PROGRAM P_UpdateDAQ
VAR_IN_OUT
	Data	: ST_DATA;
END_VAR
VAR
	DataDaq : ST_DATA;
END_VAR

DataDaq := Data;

END_PROGRAM

(* stored: Version 1.1.0.1, ProductVersion 3.1.4022.11
   POU P_UpdateDAQ: Id {13022e4a-c811-4e4c-a6ff-ab4bc1d8f568}, SpecialFunc None *)
